Universal Robots PolyScope program: IAC011 ReadID.urp

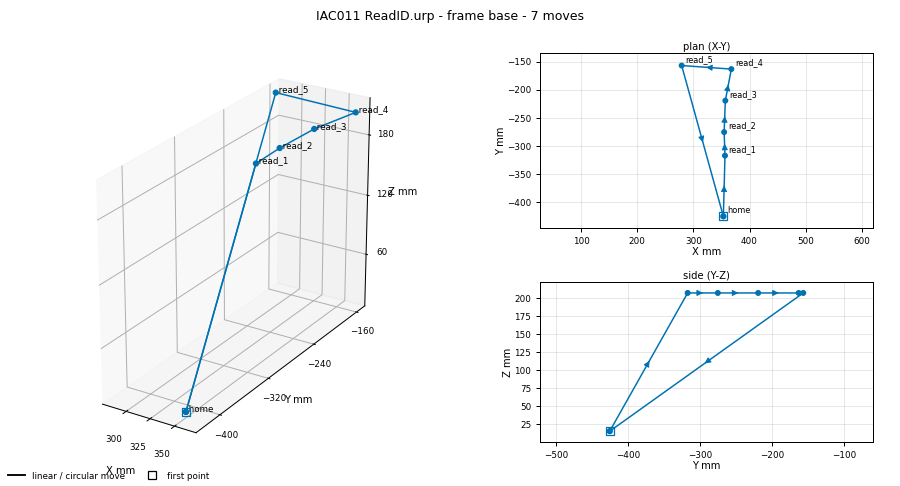
[picture p0: tool path of IAC011 ReadID.urp in frame base, 7 of 8 moves have a stored position in this frame; points joined in program order, loops and branches not executed]
Program IAC011 ReadID (installation=default directory=/programs createdIn=5.9.1.1031110 lastSavedIn=5.9.1.1031110 robotSerialNumber=20195501059)
Calibrated DH parameters: a=[0.000146, -0.418764, -0.053981, 0.000058, -0.000023, 0]; d=[0.162545, 37.319448, -206.067439, 168.881546, 0.09955, 0.099464]; alpha=[1.57004, -0.001979, 0.002304, 1.570607, -1.57066, 0]; deltaTheta=[0, -0.174616, -1.258233, 1.432844, -0.000001, 0]
BeforeStart
  URCap Gripper Activate (Robotiq_Grippers, Robotiq Inc.) dataModel(ResetAndActivateKey=false)
  initial_p := get_actual_tcp_pose()
  MoveJ speed 60 deg/s, acceleration 80 deg/s^2 (useActiveTCP=true) feature=Base
    Waypoint Waypoint (Variable): variable=initial_p
  Set DigitalOutput pin=digital_out[1]; digitalValue=1
Robot Program (runOnlyOnce=false)
  URCap Gripper (Robotiq_Grippers, Robotiq Inc.) dataModel(position=100.0, force=100.0, speed=100.0, positionInDouble=100.0, forceInDouble=100.0, speedInDouble=100.0, slaveIds=[9], blocking=true)
  MoveL speed 250 mm/s, acceleration 1200 mm/s^2 (useActiveTCP=true) feature=Base
    Waypoint home: TCP in base x=353.442 y=-425.051 z=15.364 mm, rx=-2.1827 ry=-2.2594 rz=0 rad; joints [115.734, -68.978, 112.532, -133.544, 270.037, 113.795] deg; TCP offset x=0 y=0 z=174 mm, rx=0 ry=0 rz=0 rad
  Call vision_connect
  Loop Counting (count=5) loopVariable(name=Loop_3)
    MoveL speed 250 mm/s, acceleration 1200 mm/s^2 (useActiveTCP=true) feature=Base
      Waypoint read_1: TCP in base x=356.324 y=-316.925 z=207.231 mm, rx=1.0652 ry=2.787 rz=-0.3803 rad; joints [126.838, -98.607, 119.172, -124.891, 261.973, 77.673] deg
      Call vision_read_barcode
    MoveL speed 250 mm/s, acceleration 1200 mm/s^2 (useActiveTCP=true) feature=Base
      Waypoint read_2: TCP in base x=354.825 y=-275.05 z=207.21 mm, rx=1.0911 ry=2.7792 rz=-0.3824 rad; joints [130.715, -102.216, 121.838, -123.219, 260.79, 82.491] deg
      Call vision_read_barcode
    MoveL speed 250 mm/s, acceleration 1200 mm/s^2 (useActiveTCP=true) feature=Base
      Waypoint read_3: TCP in base x=356.922 y=-219.073 z=207.206 mm, rx=1.037 ry=2.7954 rz=-0.378 rad; joints [136.698, -106.404, 124.673, -121.227, 259.917, 86.26] deg
      Call vision_read_barcode
    MoveL speed 250 mm/s, acceleration 1200 mm/s^2 (useActiveTCP=true) feature=Base
      Waypoint read_4: TCP in base x=367.655 y=-162.85 z=207.203 mm, rx=1.0723 ry=2.785 rz=-0.3809 rad; joints [145.271, -107.586, 124.958, -118.396, 257.838, 96.208] deg
      Call vision_read_barcode
    MoveL speed 250 mm/s, acceleration 1200 mm/s^2 (useActiveTCP=true) feature=Base
      Waypoint read_5: TCP in base x=279.176 y=-156.494 z=207.204 mm, rx=1.1028 ry=2.7756 rz=-0.3833 rad; joints [135.575, -123.312, 133.588, -112.971, 259.597, 87.73] deg
      Call vision_read_barcode
  MoveL speed 250 mm/s, acceleration 1200 mm/s^2 (useActiveTCP=true) feature=Base
    Waypoint home: TCP in base x=353.442 y=-425.051 z=15.364 mm, rx=-2.1827 ry=-2.2594 rz=0 rad; joints [115.734, -68.978, 112.532, -133.544, 270.037, 113.795] deg
  Call vision_disconnect
SubProgram  [hidden by the author, left out]
SubProgram  [hidden by the author, left out]
SubProgram  [hidden by the author, left out]
SubProgram vision_connect [hidden by the author, left out]
SubProgram vision_read_barcode [hidden by the author, left out]
SubProgram vision_disconnect [hidden by the author, left out]
